KUKA KRL program: FOLLOWTEST.src, FOLLOWTEST.dat

--- FOLLOWTEST.src ---
&ACCESS RVO
&REL 225
&PARAM TEMPLATE = C:\KRC\Roboter\Template\vorgabe
&PARAM EDITMASK = *
DEF FOLLOWTEST( )
INT X
DECL BOOL TEMP, SEMP, HEMP
DECL INT md_int[16]
DECL REAL md_real[16]
DECL INT n
DECL FRAME POINT
DECL INT result
;FOLD INI
  ;FOLD BASISTECH INI
    GLOBAL INTERRUPT DECL 3 WHEN $STOPMESS==TRUE DO IR_STOPM ( )
    INTERRUPT ON 3
    BAS (#INITMOV,0 )
  ;ENDFOLD (BASISTECH INI)
  ;FOLD USER INI
    ;Make your modifications here
  ;ENDFOLD (USER INI)
;ENDFOLD (INI)


$STIFFNESS.STRATEGY=10
$STIFFNESS.COMMIT=TRUE
$ORI_TYPE=#CONSTANT
$TOOL=TOOL_DATA[5]
$VEL.CP=1.0
$VEL.ORI1=100
$VEL.ORI2=100
$ACC.CP=1.0
$ACC.ORI1=100
$ACC.ORI2=100
FOR X=1 TO 6
  $ACC_AXIS[X]=100
  $VEL_AXIS[X]=100
ENDFOR
PT2={X 0,Y 0,Z 0,A 0,B 0,C 0}
$OV_PRO=40.0

;FOLD PTP P2 Vel=100 % PDAT2 Tool[5]:Pneumatic_gripper_probe Base[0];%{PE}%R 5.6.11,%MKUKATPBASIS,%CMOVE,%VPTP,%P 1:PTP, 2:P2, 3:, 5:100, 7:PDAT2
$BWDSTART=FALSE
PDAT_ACT=PPDAT2
FDAT_ACT=FP2
BAS(#PTP_PARAMS,100)
PTP XP2
;ENDFOLD

POINT=STARTPOINT(5)
PTP POINT

;IN START POINT:
;STARTPOINT(10)
;(12.30,-560.13,61.20,1.17,0,-180)
;STARTPOINT(20)
;(12.30,-560,56.38,1.17,0,-180)
;STARTPOINT(5)
;(10.73,-560,63.72,1.17,0,-180)
;STARTPOINT(15)
;(10.74,-560,59.36,1.18,0,-180)

HEMP=TRIG()
TEMP=SETSTIFF("Z",1.0)
SEMP=SETFORCE("Z",50.0)

LIN_REL{Z -5}

WAIT SEC 1

LIN_REL{Y -64}

result=MD_CMD("PAPAS","DESIREDFORCECLEAR",md_int[],md_real[])

PTP $POS_ACT_MES

$STIFFNESS.STRATEGY=10
$STIFFNESS.COMMIT=TRUE

$OV_PRO=75

LIN_REL{Z 10}

;FOLD PTP P4 Vel=100 % PDAT4 Tool[5]:Pneumatic_gripper_probe Base[0];%{PE}%R 5.6.11,%MKUKATPBASIS,%CMOVE,%VPTP,%P 1:PTP, 2:P4, 3:, 5:100, 7:PDAT4
$BWDSTART=FALSE
PDAT_ACT=PPDAT4
FDAT_ACT=FP4
BAS(#PTP_PARAMS,100)
PTP XP4
;ENDFOLD

END

--- FOLLOWTEST.dat ---
&ACCESS RVO
&REL 225
&PARAM TEMPLATE = C:\KRC\Roboter\Template\vorgabe
&PARAM EDITMASK = *
DEFDAT  FOLLOWTEST
;FOLD EXTERNAL DECLARATIONS;%{PE}%MKUKATPBASIS,%CEXT,%VCOMMON,%P
;FOLD BASISTECH EXT;%{PE}%MKUKATPBASIS,%CEXT,%VEXT,%P
EXT  BAS (BAS_COMMAND  :IN,REAL  :IN )
DECL INT SUCCESS
;ENDFOLD (BASISTECH EXT)
;FOLD USER EXT;%{E}%MKUKATPUSER,%CEXT,%VEXT,%P
;Make here your modifications

;ENDFOLD (USER EXT)
;ENDFOLD (EXTERNAL DECLARATIONS)
DECL BASIS_SUGG_T LAST_BASIS={POINT1[] "P4                      ",POINT2[] "P4                      ",CP_PARAMS[] "CPDAT0                  ",PTP_PARAMS[] "PDAT4                   ",CONT[] "                        ",CP_VEL[] "2.0                     ",PTP_VEL[] "100                     ",SYNC_PARAMS[] "SYNCDAT                 ",SPL_NAME[] "S0                      "}
DECL E6POS XP1={X 12.30863,Y -591.564026,Z 156.116104,A 1.18070102,B -0.00134391699,C -179.9702,S 1,T 36,E1 -0.0126686096,E2 0.0,E3 0.0,E4 0.0,E5 0.0,E6 0.0}
DECL FDAT FP1={TOOL_NO 5,BASE_NO 0,IPO_FRAME #BASE,POINT2[] " ",TQ_STATE FALSE}
DECL PDAT PPDAT1={VEL 100.0,ACC 100.0,APO_DIST 100.0,APO_MODE #CPTP}
DECL E6POS XP2={X 12.3066502,Y -560.418701,Z 81.0944366,A 1.16489899,B -0.00030443311,C -179.937698,S 1,T 36,E1 -0.0103941001,E2 0.0,E3 0.0,E4 0.0,E5 0.0,E6 0.0}
DECL FDAT FP2={TOOL_NO 5,BASE_NO 0,IPO_FRAME #BASE,POINT2[] " ",TQ_STATE FALSE}
DECL PDAT PPDAT2={VEL 100.0,ACC 100.0,APO_DIST 100.0,APO_MODE #CPTP}
DECL E6POS XP3={X 10.7449903,Y -560.32489,Z 59.3970795,A 1.174896,B 0.00173025299,C -179.957993,S 1,T 36,E1 -0.0109090796,E2 0.0,E3 0.0,E4 0.0,E5 0.0,E6 0.0}
DECL FDAT FP3={TOOL_NO 5,BASE_NO 0,IPO_FRAME #BASE,POINT2[] " ",TQ_STATE FALSE}
DECL PDAT PPDAT3={VEL 100.0,ACC 100.0,APO_DIST 100.0,APO_MODE #CPTP}
DECL INT LAST_XP_POINT=3
DECL E6POS XP4={X 12.3066502,Y -560.418701,Z 81.0944366,A 1.16489899,B -0.00030443311,C -179.937698,S 1,T 36,E1 -0.0103941001,E2 0.0,E3 0.0,E4 0.0,E5 0.0,E6 0.0}
DECL FDAT FP4={TOOL_NO 5,BASE_NO 0,IPO_FRAME #BASE,POINT2[] " ",TQ_STATE FALSE}
DECL PDAT PPDAT4={VEL 100.0,ACC 100.0,APO_DIST 100.0,APO_MODE #CPTP}
ENDDAT
